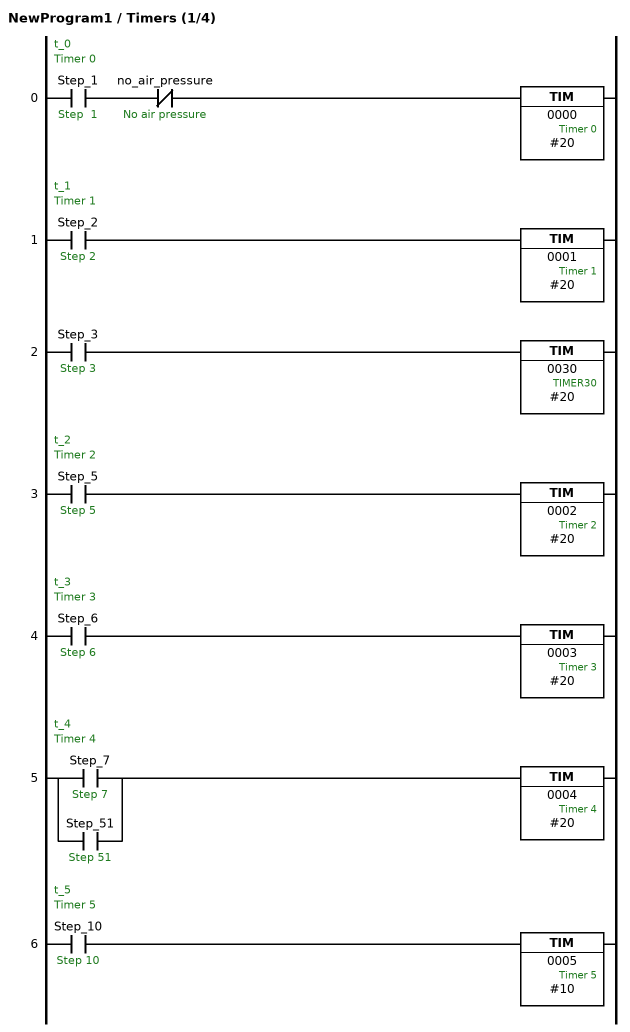
; [picture p24: NewProgram1 / Timers, rungs 0-6]
; rung 0: t_0 / Timer 0
LD Step_1  ; Step  1
ANDNOT no_air_pressure  ; No air pressure
TIM 0000 #20  ; Timer 0
; rung 1: t_1 / Timer 1
LD Step_2  ; Step 2
TIM 0001 #20  ; Timer 1
; rung 2
LD Step_3  ; Step 3
TIM 0030 #20  ; TIMER30
; rung 3: t_2 / Timer 2
LD Step_5  ; Step 5
TIM 0002 #20  ; Timer 2
; rung 4: t_3 / Timer 3
LD Step_6  ; Step 6
TIM 0003 #20  ; Timer 3
; rung 5: t_4 / Timer 4
LD Step_7  ; Step 7
OR Step_51  ; Step 51
TIM 0004 #20  ; Timer 4
; rung 6: t_5 / Timer 5
LD Step_10  ; Step 10
TIM 0005 #10  ; Timer 5

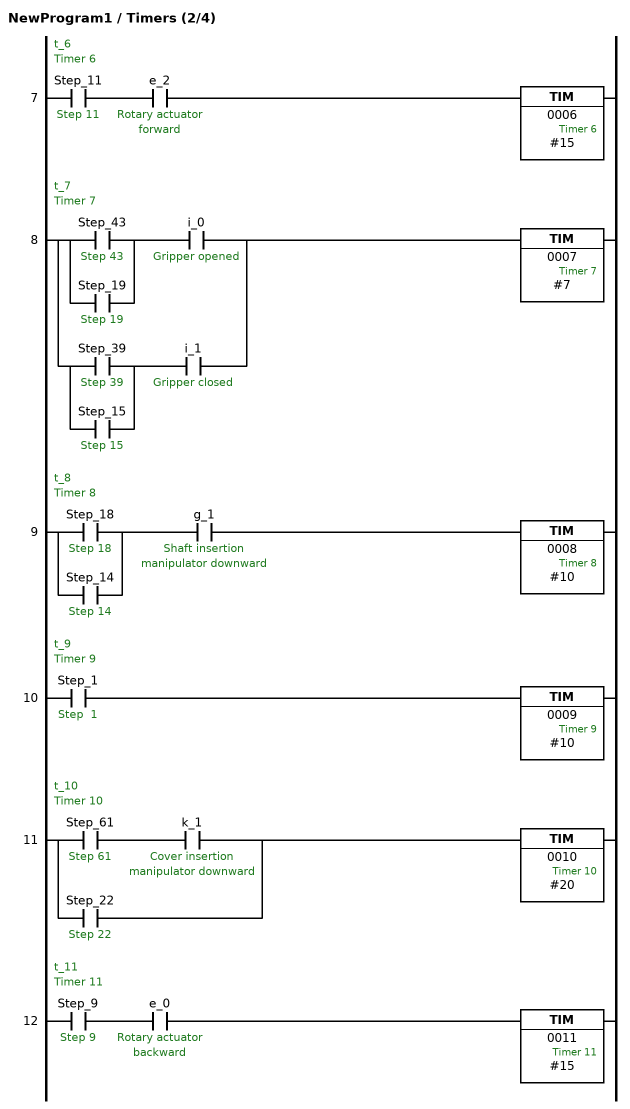
; rung 7: t_6 / Timer 6
LD Step_11  ; Step 11
AND e_2  ; Rotary actuator forward
TIM 0006 #15  ; Timer 6
; rung 8: t_7 / Timer 7
LD Step_43  ; Step 43
OR Step_19  ; Step 19
AND i_0  ; Gripper opened
LD Step_39  ; Step 39
OR Step_15  ; Step 15
AND i_1  ; Gripper closed
ORLD
TIM 0007 #7  ; Timer 7
; rung 9: t_8 / Timer 8
LD Step_18  ; Step 18
OR Step_14  ; Step 14
AND g_1  ; Shaft insertion manipulator downward
TIM 0008 #10  ; Timer 8
; rung 10: t_9 / Timer 9
LD Step_1  ; Step  1
TIM 0009 #10  ; Timer 9
; rung 11: t_10 / Timer 10
LD Step_61  ; Step 61
AND k_1  ; Cover insertion manipulator downward
OR Step_22  ; Step 22
TIM 0010 #20  ; Timer 10
; rung 12: t_11 / Timer 11
LD Step_9  ; Step 9
AND e_0  ; Rotary actuator backward
TIM 0011 #15  ; Timer 11

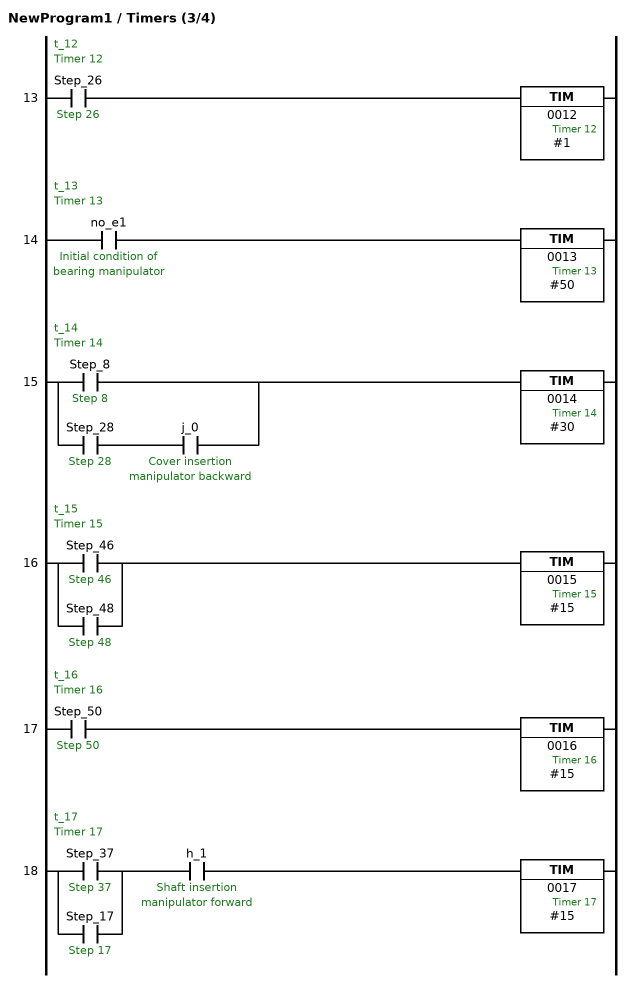
; rung 13: t_12 / Timer 12
LD Step_26  ; Step 26
TIM 0012 #1  ; Timer 12
; rung 14: t_13 / Timer 13
LD no_e1  ; Initial condition of bearing manipulator
TIM 0013 #50  ; Timer 13
; rung 15: t_14 / Timer 14
LD Step_8  ; Step 8
LD Step_28  ; Step 28
AND j_0  ; Cover insertion manipulator backward
ORLD
TIM 0014 #30  ; Timer 14
; rung 16: t_15 / Timer 15
LD Step_46  ; Step 46
OR Step_48  ; Step 48
TIM 0015 #15  ; Timer 15
; rung 17: t_16 / Timer 16
LD Step_50  ; Step 50
TIM 0016 #15  ; Timer 16
; rung 18: t_17 / Timer 17
LD Step_37  ; Step 37
OR Step_17  ; Step 17
AND h_1  ; Shaft insertion manipulator forward
TIM 0017 #15  ; Timer 17

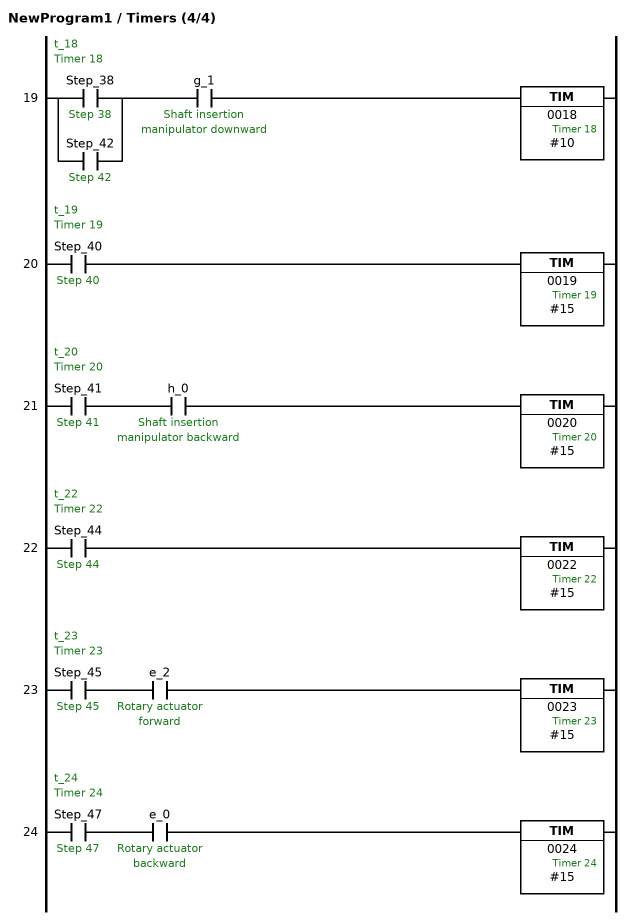
; rung 19: t_18 / Timer 18
LD Step_38  ; Step 38
OR Step_42  ; Step 42
AND g_1  ; Shaft insertion manipulator downward
TIM 0018 #10  ; Timer 18
; rung 20: t_19 / Timer 19
LD Step_40  ; Step 40
TIM 0019 #15  ; Timer 19
; rung 21: t_20 / Timer 20
LD Step_41  ; Step 41
AND h_0  ; Shaft insertion manipulator backward
TIM 0020 #15  ; Timer 20
; rung 22: t_22 / Timer 22
LD Step_44  ; Step 44
TIM 0022 #15  ; Timer 22
; rung 23: t_23 / Timer 23
LD Step_45  ; Step 45
AND e_2  ; Rotary actuator forward
TIM 0023 #15  ; Timer 23
; rung 24: t_24 / Timer 24
LD Step_47  ; Step 47
AND e_0  ; Rotary actuator backward
TIM 0024 #15  ; Timer 24

### Section Cover_detection

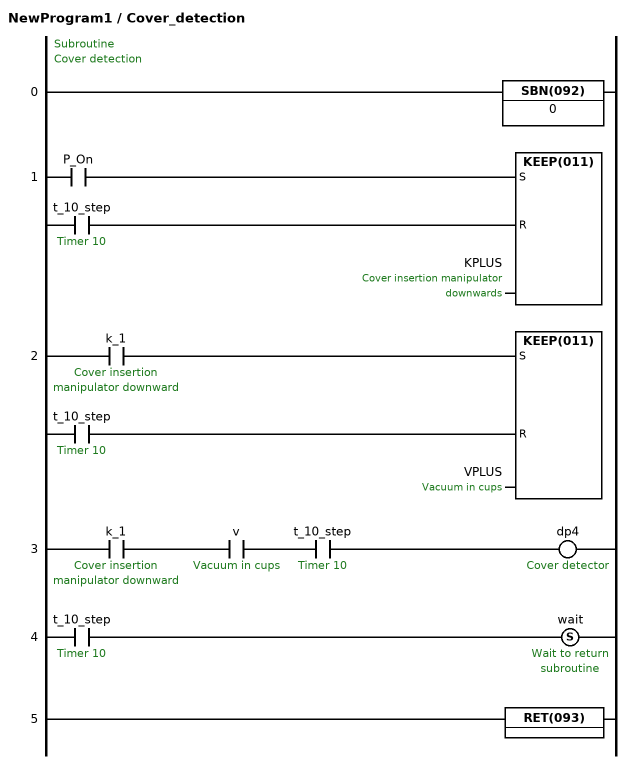
; rung 0: Subroutine / Cover detection
SBN(092) 0
; rung 1
LD P_On
LD t_10_step  ; Timer 10
KEEP(011) KPLUS  ; Cover insertion manipulator downwards
; rung 2
LD k_1  ; Cover insertion manipulator downward
LD t_10_step  ; Timer 10
KEEP(011) VPLUS  ; Vacuum in cups
; rung 3
LD k_1  ; Cover insertion manipulator downward
AND v  ; Vacuum in cups
AND t_10_step  ; Timer 10
OUT dp4  ; Cover detector
; rung 4
LD t_10_step  ; Timer 10
SET wait  ; Wait to return subroutine
; rung 5
RET(093)
; rung 6
END(001)